(* PLC project Generated.project, CODESYS CODESYS V3.5 SP19 Patch 1 *)
(* stored: creationDateTime 2026-09-06T13:00:42.407428, modificationDateTime 2026-09-06T13:00:42.407428 *)

(* values of E_OperatorAxis: NONE: Aucun axe attendu (étape automatique ou arrêt); JOYSTICK_X: Axe X translation attendu; JOYSTICK_Y: Axe Y treuils / plongée attendu; BUTTON: Action bouton attendue (ex: validation, homing) *)

{attribute 'qualified_only'}
{attribute 'strict'}
TYPE E_OperatorAxis : (NONE := 0, JOYSTICK_X := 1, JOYSTICK_Y := 2, BUTTON := 3);
END_TYPE
